// TwinCAT 3 PLC project PLC
// ProgramVersion: 3.1.4026.19
// libraries:
//   Tc2_MC2, * (Beckhoff Automation GmbH)
//   Tc2_Standard, * (Beckhoff Automation GmbH)
//   Tc2_System, * (Beckhoff Automation GmbH)
// project tree:
//   / PlcTask.TcTTO
//   POUs/ MAIN.TcPOU
// real-time tasks:
//   TASK PlcTask: cycle T#10ms, priority 20, ADS port 350
// motion (NC):
//   TASK NC-Task 1 SAF: cycle T#2ms, priority 4, ADS port 501
//   TASK NC-Task 1 SVB: cycle T#10ms, priority 8, ADS port 511
//   AXIS Axis 1 (id 1)
//     OtherSettings: AllowMotionCmdToSlave=true
//     encoder EncType=1
//     drive DrvType=5
//       Analog: TorqueSetpointScale=10, ScaleFactorActTorque=0.1
//     controller CtrType=1
//       CtrPara: PriorControlFactor=1
//         Observer: BandWidth=20
// variable links:
//   PLC/PLC Instance <-> NC-Task 1 SAF/Axes/Axis 1
//     PlcTask Inputs/MAIN.axisVirtualMotor.NcToPlc <-> Outputs/ToPlc
//     PlcTask Outputs/MAIN.axisVirtualMotor.PlcToNc <-> Inputs/FromPlc

CONFIGURATION PLC
    RESOURCE PLC ON TwinCAT3
        TASK PlcTask(INTERVAL := T#10ms, PRIORITY := 20);
        PROGRAM MAIN WITH PlcTask : MAIN;
    END_RESOURCE
END_CONFIGURATION

// ---- POUs/MAIN.TcPOU
PROGRAM MAIN
VAR
    axisVirtualMotor : AXIS_REF; 
    
    fbPower : MC_Power;
    bEnable : BOOL := TRUE;    

    fbMove  : MC_MoveAbsolute;
    bExecuteMove : BOOL;        
    fTargetPosition : LREAL;     

    iState      : INT := 0;     
    bAutoStart  : BOOL;        
    fbWaitTimer : TON;           
END_VAR

fbPower(
    Axis := axisVirtualMotor,
    Enable := bEnable,
    Enable_Positive := bEnable,
    Enable_Negative := bEnable,
    Override := 100.0
);


fbMove(
    Axis := axisVirtualMotor,
    Execute := bExecuteMove,
    Position := fTargetPosition,
    Velocity := 100.0
);


fbWaitTimer(IN := (iState = 20), PT := T#2S);


CASE iState OF
    
    0: 
        bExecuteMove := FALSE; 
        IF bAutoStart THEN
            bAutoStart := FALSE;      
            fTargetPosition := 150.5; 
            bExecuteMove := TRUE;     
            iState := 10;             
        END_IF
        
    10: 
        IF fbMove.Done THEN      
            bExecuteMove := FALSE;    
            iState := 20;             
        END_IF
        
    20: 
        IF fbWaitTimer.Q THEN         
            fTargetPosition := 0.0;  
            bExecuteMove := TRUE;    
            iState := 30;             
        END_IF
        
    30: 
        IF fbMove.Done THEN           
            bExecuteMove := FALSE;    
            iState := 0;              
        END_IF

END_CASE

END_PROGRAM
